# EPICS substitutions: NEOCERA/NEOCERA-IOC-01App/Db/unit_setter.substitutions
# Set points do not have units set because it will cause it to be processed thus sending a possibly wrong value
# to the display

file $(UTILITIES)/db/unit_setter.template {
  pattern
    {P,    FROM, TO}

    {"\$(P)", "1:TEMP:UNITS", "1:TEMP"}
	{"\$(P)", "2:TEMP:UNITS", "2:TEMP"}
	{"\$(P)", "1:TEMP:SP:UNITS", "1:TEMP:SP:RBV"}
	{"\$(P)", "2:TEMP:SP:UNITS", "2:TEMP:SP:RBV"}
}
